Fanuc KAREL source: IO0034.KL

PROGRAM IO0034
%STACKSIZE=65535
%PRIORITY=65535
%NOLOCKGROUP
ROUTINE RTEST FROM IO0034
ROUTINE RTEST
VAR
L1 : ARRAY[3] OF INTEGER
L2 : XYZWPR
L3 : JOINTPOS9
L4 : POSITION
U2C_37 : INTEGER
U2C_38 : REAL
U2C_39 : REAL
U2C_40 : INTEGER
U2C_41 : REAL
BEGIN
U2C_37=1
L1[1]=2
U2C_40=1
U2C_41=1.0
DOUT[L1[U2C_37]]=U2C_40
END RTEST
BEGIN
RTEST
END IO0034
